FUNCTION_BLOCK IF_selfmade (* Composite Function Block Type *)
  (* Standard: 61499-2 *)
  (* Version 0.2, 2003-12-05, JHC, Rockwell Automation, Renamed from NEWCOMPFB. *)
  (* Version 0.1, 2002-01-08, JHC, Rockwell Automation, Added DLY FB as example. *)
  (* Version 0.0, 2000-05-27, JHC, Rockwell Automation *)
  (* Compiler header: package fb.rt.template; *)
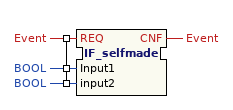
  EVENT_INPUT
    REQ WITH Input1, input2; (* Normal Execution Request *)
  END_EVENT
  EVENT_OUTPUT
    CNF; (* Execution Confirmation *)
  END_EVENT
  VAR_INPUT
    Input1 : BOOL;
    input2 : BOOL;
  END_VAR
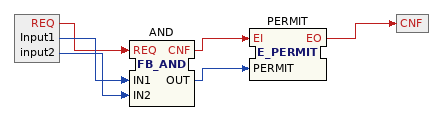
  FBS
    AND : FB_AND;
    PERMIT : E_PERMIT;
  END_FBS
  EVENT_CONNECTIONS
    REQ TO AND.REQ;
    AND.CNF TO PERMIT.EI;
    PERMIT.EO TO CNF;
  END_CONNECTIONS
  DATA_CONNECTIONS
    Input1 TO AND.IN1;
    input2 TO AND.IN2;
    AND.OUT TO PERMIT.PERMIT;
  END_CONNECTIONS
END_FUNCTION_BLOCK
